Universal Robots PolyScope program: taskboard_place_hook.urp

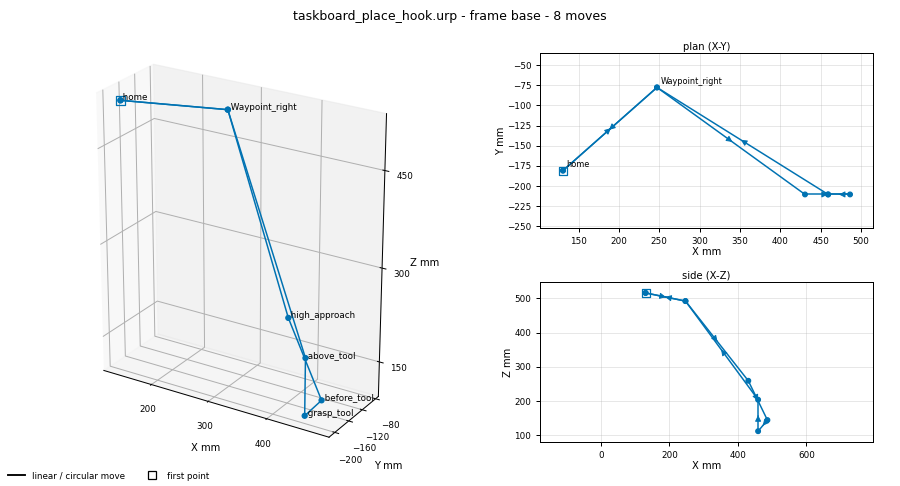
[picture p0: tool path of taskboard_place_hook.urp in frame base, 8 of 9 moves have a stored position in this frame; points joined in program order, loops and branches not executed]
Program taskboard_place_hook (installation=default directory=/programs/wrs2020 createdIn=5.10.0.106288 lastSavedIn=5.10.0.106288 robotSerialNumber=20205500607)
Calibrated DH parameters: a=[0.000096, -0.337, -0.383372, 0.000118, 0.000015, 0]; d=[0.162724, 79.377998, -95.545185, 16.300583, 0.099689, 0.099499]; alpha=[1.569249, 0.003272, 0.005201, 1.570041, -1.570219, 0]; deltaTheta=[0, 0.65664, 5.410619, 0.215927, -0.000001, 0]
Robot Program (runOnlyOnce=true)
  MoveJ speed 60 deg/s, acceleration 80 deg/s^2 (useActiveTCP=true) feature=Base
    currentpose := get_actual_joint_positions()
    Waypoint Waypoint (Variable): variable=currentpose
  MoveL speed 1200 mm/s, acceleration 800 mm/s^2 (useActiveTCP=false) tcp=TCP; feature=Base
    Waypoint home: TCP in base x=130.649 y=-180.735 z=515.945 mm, rx=-0.0119 ry=-3.1403 rz=-0.0318 rad; joints [89.95, -120.316, 80.212, -48.703, -89.953, 0.003] deg; TCP offset x=0 y=0 z=165 mm, rx=0 ry=0 rz=0 rad
    Waypoint Waypoint_right: motionParameters(blendRadius=0.05); TCP in base x=247.136 y=-77.743 z=492.156 mm, rx=-1.0893 ry=2.9411 rz=0.0437 rad; joints [131.739, -127.117, 113.467, -74.929, -88.981, 0.805] deg
    Waypoint high_approach: motionParameters(blendRadius=0.05); TCP in base x=430.518 y=-210.304 z=259.484 mm, rx=2.0705 ry=-2.0633 rz=-0.2652 rad; joints [140.289, -82.581, 114.687, -110.586, -100.48, -38.868] deg
    Waypoint before_tool: motionParameters(blendRadius=0.005); TCP in base x=486.311 y=-210.304 z=144.711 mm, rx=1.7463 ry=-1.7306 rz=-0.729 rad; joints [146.732, -60.807, 101.299, -89.72, -114.09, -24.722] deg
    Waypoint grasp_tool: TCP in base x=459.162 y=-210.304 z=112.252 mm, rx=1.7463 ry=-1.7306 rz=-0.729 rad; joints [145.194, -60.295, 107.111, -96.572, -115.081, -25.972] deg
    URCap Gripper (Robotiq_Grippers, Robotiq Inc.) dataModel(position=0.0, force=100.0, speed=100.0, positionInDouble=0.0, forceInDouble=100.0, speedInDouble=100.0, slaveIds=[9], blocking=true)
    Waypoint above_tool: motionParameters(blendRadius=0.01); TCP in base x=459.162 y=-210.304 z=204.201 mm, rx=1.7463 ry=-1.7306 rz=-0.729 rad; joints [145.218, -68.652, 102.912, -84.042, -115.104, -26.034] deg
    Waypoint Waypoint_right: motionParameters(blendRadius=0.05); TCP in base x=247.136 y=-77.743 z=492.156 mm, rx=-1.0893 ry=2.9411 rz=0.0437 rad; joints [131.739, -127.117, 113.467, -74.929, -88.981, 0.805] deg
    Waypoint home: TCP in base x=130.649 y=-180.735 z=515.945 mm, rx=-0.0119 ry=-3.1403 rz=-0.0318 rad; joints [89.95, -120.316, 80.212, -48.703, -89.953, 0.003] deg; TCP offset x=0 y=0 z=165 mm, rx=0 ry=0 rz=0 rad
